{attribute 'qualified_only'}
{attribute 'strict'}
TYPE AutostoreStatus :
(
	UNKNOWN := 0,
	EXCHANGING	:=1,
	READY	:=2
);
END_TYPE

(* stored: Version 1.1.0.1, ProductVersion 3.1.4024.12
   DUT AutostoreStatus: Id {b67a0d6e-0dc7-4cb5-94de-8340c9efb89c} *)
